// TIA Portal V20 export
FUNCTION "04 T1-A ARUNC Transitions" : Void   // FC1402, LAD
TITLE = TRANSITIONS
{ S7_Optimized_Access := 'TRUE' }
// stored: AutoNumber false, SetENOAutomatically false
   VAR_TEMP
      Aux_real : Real;
   END_VAR
BEGIN

REGION Network 1: ============ TRANSITIONS ============
END_REGION

REGION Network 2: Transitions - Zone Status
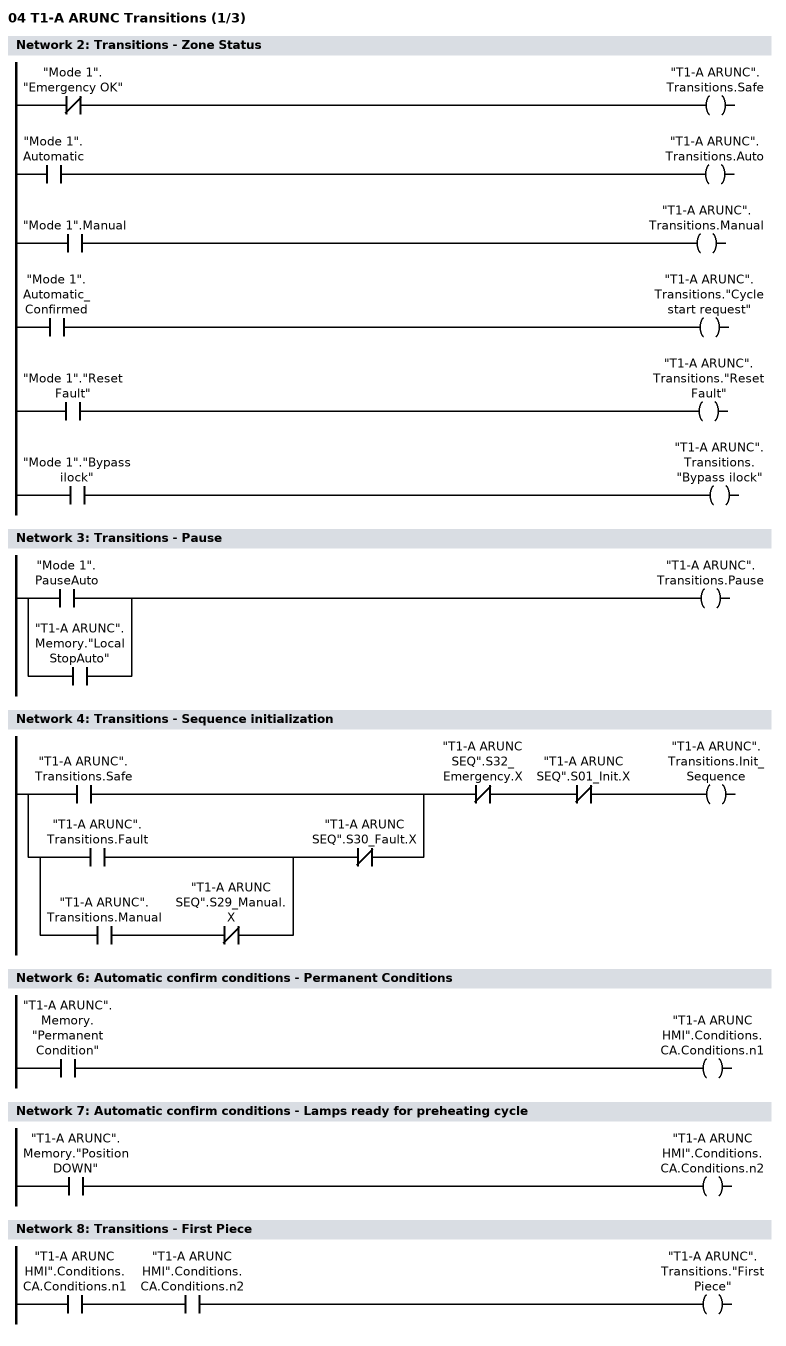
   RUNG wire#powerrail
      I_Contact( "Mode 1"."Emergency OK" )
      Coil( "T1-A ARUNC".Transitions.Safe )
   END_RUNG
   RUNG wire#powerrail
      Contact( "Mode 1".Automatic )
      Coil( "T1-A ARUNC".Transitions.Auto )
   END_RUNG
   RUNG wire#powerrail
      Contact( "Mode 1".Manual )
      Coil( "T1-A ARUNC".Transitions.Manual )
   END_RUNG
   RUNG wire#powerrail
      Contact( "Mode 1".Automatic_Confirmed )
      Coil( "T1-A ARUNC".Transitions."Cycle start request" )
   END_RUNG
   RUNG wire#powerrail
      Contact( "Mode 1"."Reset Fault" )
      Coil( "T1-A ARUNC".Transitions."Reset Fault" )
   END_RUNG
   RUNG wire#powerrail
      Contact( "Mode 1"."Bypass ilock" )
      Coil( "T1-A ARUNC".Transitions."Bypass ilock" )
   END_RUNG
   // the same network as SCL:
   "T1-A ARUNC".Transitions.Safe := NOT "Mode 1"."Emergency OK";
   "T1-A ARUNC".Transitions.Auto := "Mode 1".Automatic;
   "T1-A ARUNC".Transitions.Manual := "Mode 1".Manual;
   "T1-A ARUNC".Transitions."Cycle start request" := "Mode 1".Automatic_Confirmed;
   "T1-A ARUNC".Transitions."Reset Fault" := "Mode 1"."Reset Fault";
   "T1-A ARUNC".Transitions."Bypass ilock" := "Mode 1"."Bypass ilock";
END_REGION

REGION Network 3: Transitions - Pause
   RUNG wire#powerrail
      Contact( "Mode 1".PauseAuto )
      wire#w1
      Coil( "T1-A ARUNC".Transitions.Pause )
   END_RUNG
   RUNG wire#powerrail
      Contact( "T1-A ARUNC".Memory."Local StopAuto" )
   END_RUNG wire#w1
   // the same network as SCL:
   "T1-A ARUNC".Transitions.Pause := "Mode 1".PauseAuto OR "T1-A ARUNC".Memory."Local StopAuto";
END_REGION

REGION Network 4: Transitions - Sequence initialization
   RUNG wire#powerrail
      Contact( "T1-A ARUNC".Transitions.Safe )
      wire#w1
      I_Contact( "T1-A ARUNC SEQ".S32_Emergency.X )
      I_Contact( "T1-A ARUNC SEQ".S01_Init.X )
      Coil( "T1-A ARUNC".Transitions.Init_Sequence )
   END_RUNG
   RUNG wire#powerrail
      Contact( "T1-A ARUNC".Transitions.Fault )
      wire#w2
      I_Contact( "T1-A ARUNC SEQ".S30_Fault.X )
   END_RUNG wire#w1
   RUNG wire#powerrail
      Contact( "T1-A ARUNC".Transitions.Manual )
      I_Contact( "T1-A ARUNC SEQ".S29_Manual.X )
   END_RUNG wire#w2
   // the same network as SCL:
   "T1-A ARUNC".Transitions.Init_Sequence := ("T1-A ARUNC".Transitions.Safe OR (("T1-A ARUNC".Transitions.Fault OR ("T1-A ARUNC".Transitions.Manual AND NOT "T1-A ARUNC SEQ".S29_Manual.X)) AND NOT "T1-A ARUNC SEQ".S30_Fault.X)) AND NOT "T1-A ARUNC SEQ".S32_Emergency.X AND NOT "T1-A ARUNC SEQ".S01_Init.X;
END_REGION

REGION Network 5: ============ AUTOMATIC CONFIRM CONDITIONS - 1ST PIECE ============
END_REGION

REGION Network 6: Automatic confirm conditions - Permanent Conditions
   RUNG wire#powerrail
      Contact( "T1-A ARUNC".Memory."Permanent Condition" )
      Coil( "T1-A ARUNC HMI".Conditions.CA.Conditions.n1 )
   END_RUNG
   // the same network as SCL:
   "T1-A ARUNC HMI".Conditions.CA.Conditions.n1 := "T1-A ARUNC".Memory."Permanent Condition";
END_REGION

REGION Network 7: Automatic confirm conditions - Lamps ready for preheating cycle
   RUNG wire#powerrail
      Contact( "T1-A ARUNC".Memory."Position DOWN" )
      Coil( "T1-A ARUNC HMI".Conditions.CA.Conditions.n2 )
   END_RUNG
   // the same network as SCL:
   "T1-A ARUNC HMI".Conditions.CA.Conditions.n2 := "T1-A ARUNC".Memory."Position DOWN";
END_REGION

REGION Network 8: Transitions - First Piece
   RUNG wire#powerrail
      Contact( "T1-A ARUNC HMI".Conditions.CA.Conditions.n1 )
      Contact( "T1-A ARUNC HMI".Conditions.CA.Conditions.n2 )
      Coil( "T1-A ARUNC".Transitions."First Piece" )
   END_RUNG
   // the same network as SCL:
   "T1-A ARUNC".Transitions."First Piece" := "T1-A ARUNC HMI".Conditions.CA.Conditions.n1 AND "T1-A ARUNC HMI".Conditions.CA.Conditions.n2;
END_REGION

REGION Network 9: Transitions - Piece presence
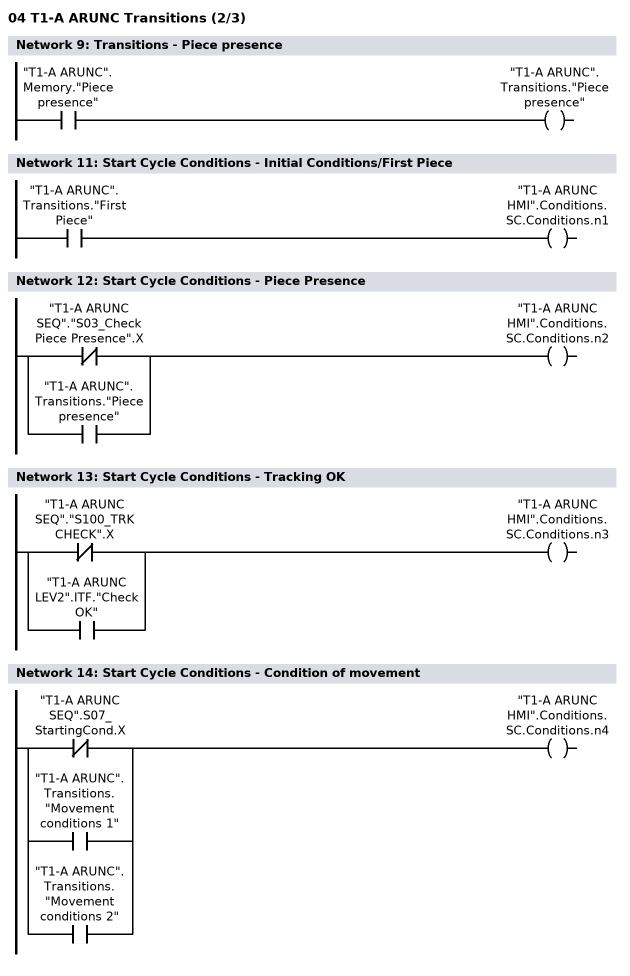
   RUNG wire#powerrail
      Contact( "T1-A ARUNC".Memory."Piece presence" )
      Coil( "T1-A ARUNC".Transitions."Piece presence" )
   END_RUNG
   // the same network as SCL:
   "T1-A ARUNC".Transitions."Piece presence" := "T1-A ARUNC".Memory."Piece presence";
END_REGION

REGION Network 10: ============ START CYCLE CONDITIONS ============
END_REGION

REGION Network 11: Start Cycle Conditions - Initial Conditions/First Piece
   RUNG wire#powerrail
      Contact( "T1-A ARUNC".Transitions."First Piece" )
      Coil( "T1-A ARUNC HMI".Conditions.SC.Conditions.n1 )
   END_RUNG
   // the same network as SCL:
   "T1-A ARUNC HMI".Conditions.SC.Conditions.n1 := "T1-A ARUNC".Transitions."First Piece";
END_REGION

REGION Network 12: Start Cycle Conditions - Piece Presence
   RUNG wire#powerrail
      I_Contact( "T1-A ARUNC SEQ"."S03_Check Piece Presence".X )
      wire#w1
      Coil( "T1-A ARUNC HMI".Conditions.SC.Conditions.n2 )
   END_RUNG
   RUNG wire#powerrail
      Contact( "T1-A ARUNC".Transitions."Piece presence" )
   END_RUNG wire#w1
   // the same network as SCL:
   "T1-A ARUNC HMI".Conditions.SC.Conditions.n2 := NOT "T1-A ARUNC SEQ"."S03_Check Piece Presence".X OR "T1-A ARUNC".Transitions."Piece presence";
END_REGION

REGION Network 13: Start Cycle Conditions - Tracking OK
   RUNG wire#powerrail
      I_Contact( "T1-A ARUNC SEQ"."S100_TRK CHECK".X )
      wire#w1
      Coil( "T1-A ARUNC HMI".Conditions.SC.Conditions.n3 )
   END_RUNG
   RUNG wire#powerrail
      Contact( "T1-A ARUNC LEV2".ITF."Check OK" )
   END_RUNG wire#w1
   // the same network as SCL:
   "T1-A ARUNC HMI".Conditions.SC.Conditions.n3 := NOT "T1-A ARUNC SEQ"."S100_TRK CHECK".X OR "T1-A ARUNC LEV2".ITF."Check OK";
END_REGION

REGION Network 14: Start Cycle Conditions - Condition of movement
   RUNG wire#powerrail
      I_Contact( "T1-A ARUNC SEQ".S07_StartingCond.X )
      wire#w1
      Coil( "T1-A ARUNC HMI".Conditions.SC.Conditions.n4 )
   END_RUNG
   RUNG wire#powerrail
      Contact( "T1-A ARUNC".Transitions."Movement conditions 1" )
   END_RUNG wire#w1
   RUNG wire#powerrail
      Contact( "T1-A ARUNC".Transitions."Movement conditions 2" )
   END_RUNG wire#w1
   // the same network as SCL:
   "T1-A ARUNC HMI".Conditions.SC.Conditions.n4 := NOT "T1-A ARUNC SEQ".S07_StartingCond.X OR "T1-A ARUNC".Transitions."Movement conditions 1" OR "T1-A ARUNC".Transitions."Movement conditions 2";
END_REGION

REGION Network 15: Start Cycle Conditions - next machine consent
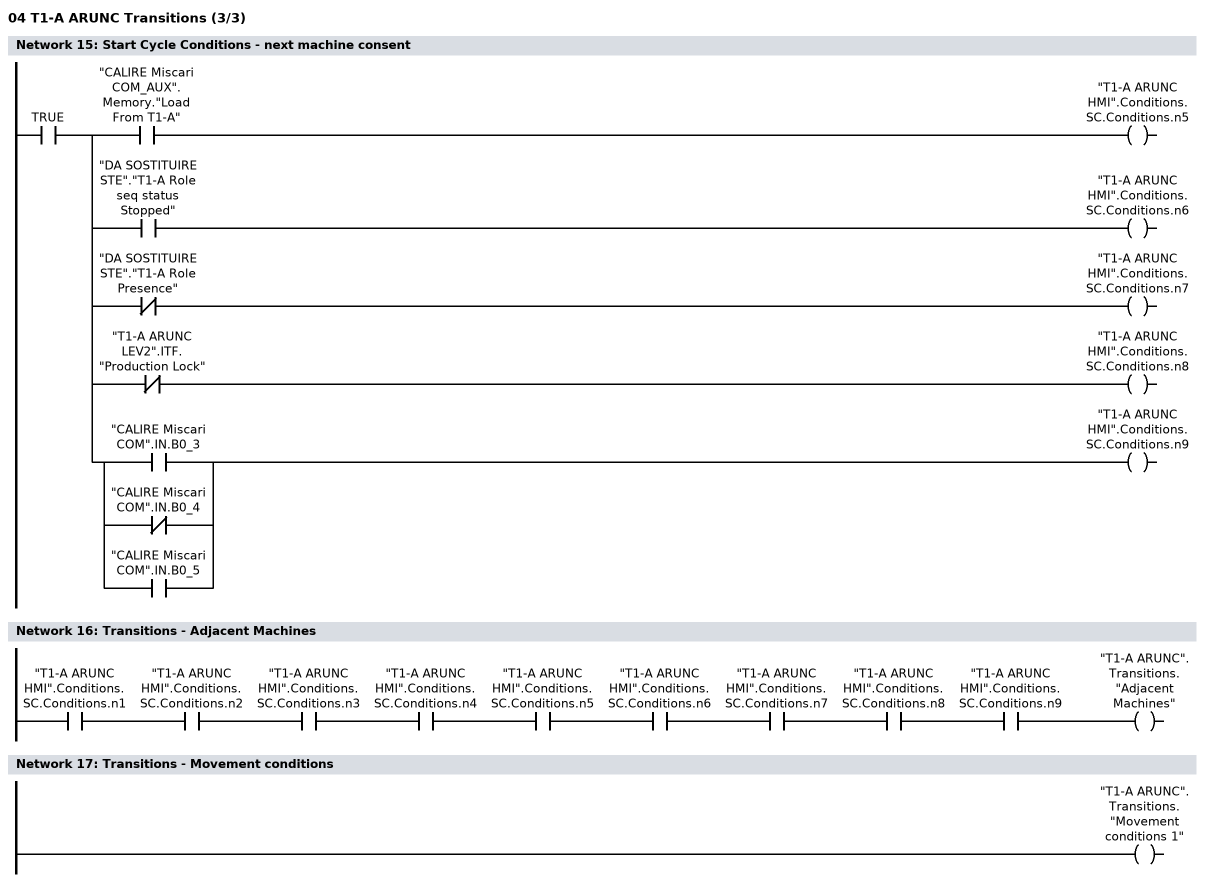
   RUNG wire#powerrail
      Contact( TRUE )
      wire#w1
      Contact( "CALIRE Miscari COM_AUX".Memory."Load From T1-A" )
      Coil( "T1-A ARUNC HMI".Conditions.SC.Conditions.n5 )
   END_RUNG
   RUNG wire#w1
      Contact( "DA SOSTITUIRE STE"."T1-A Role seq status Stopped" )
      Coil( "T1-A ARUNC HMI".Conditions.SC.Conditions.n6 )
   END_RUNG
   RUNG wire#w1
      I_Contact( "DA SOSTITUIRE STE"."T1-A Role Presence" )
      Coil( "T1-A ARUNC HMI".Conditions.SC.Conditions.n7 )
   END_RUNG
   RUNG wire#w1
      I_Contact( "T1-A ARUNC LEV2".ITF."Production Lock" )
      Coil( "T1-A ARUNC HMI".Conditions.SC.Conditions.n8 )
   END_RUNG
   RUNG wire#w1
      Contact( "CALIRE Miscari COM".IN.B0_3 )
      wire#w2
      Coil( "T1-A ARUNC HMI".Conditions.SC.Conditions.n9 )
   END_RUNG
   RUNG wire#w1
      I_Contact( "CALIRE Miscari COM".IN.B0_4 )
   END_RUNG wire#w2
   RUNG wire#w1
      Contact( "CALIRE Miscari COM".IN.B0_5 )
   END_RUNG wire#w2
   // the same network as SCL:
   "T1-A ARUNC HMI".Conditions.SC.Conditions.n5 := TRUE AND "CALIRE Miscari COM_AUX".Memory."Load From T1-A";
   "T1-A ARUNC HMI".Conditions.SC.Conditions.n6 := TRUE AND "DA SOSTITUIRE STE"."T1-A Role seq status Stopped";
   "T1-A ARUNC HMI".Conditions.SC.Conditions.n7 := TRUE AND NOT "DA SOSTITUIRE STE"."T1-A Role Presence";
   "T1-A ARUNC HMI".Conditions.SC.Conditions.n8 := TRUE AND NOT "T1-A ARUNC LEV2".ITF."Production Lock";
   "T1-A ARUNC HMI".Conditions.SC.Conditions.n9 := TRUE AND ("CALIRE Miscari COM".IN.B0_3 OR NOT "CALIRE Miscari COM".IN.B0_4 OR "CALIRE Miscari COM".IN.B0_5);
END_REGION

REGION Network 16: Transitions - Adjacent Machines
   RUNG wire#powerrail
      Contact( "T1-A ARUNC HMI".Conditions.SC.Conditions.n1 )
      Contact( "T1-A ARUNC HMI".Conditions.SC.Conditions.n2 )
      Contact( "T1-A ARUNC HMI".Conditions.SC.Conditions.n3 )
      Contact( "T1-A ARUNC HMI".Conditions.SC.Conditions.n4 )
      Contact( "T1-A ARUNC HMI".Conditions.SC.Conditions.n5 )
      Contact( "T1-A ARUNC HMI".Conditions.SC.Conditions.n6 )
      Contact( "T1-A ARUNC HMI".Conditions.SC.Conditions.n7 )
      Contact( "T1-A ARUNC HMI".Conditions.SC.Conditions.n8 )
      Contact( "T1-A ARUNC HMI".Conditions.SC.Conditions.n9 )
      Coil( "T1-A ARUNC".Transitions."Adjacent Machines" )
   END_RUNG
   // the same network as SCL:
   "T1-A ARUNC".Transitions."Adjacent Machines" := "T1-A ARUNC HMI".Conditions.SC.Conditions.n1 AND "T1-A ARUNC HMI".Conditions.SC.Conditions.n2 AND "T1-A ARUNC HMI".Conditions.SC.Conditions.n3 AND "T1-A ARUNC HMI".Conditions.SC.Conditions.n4 AND "T1-A ARUNC HMI".Conditions.SC.Conditions.n5 AND "T1-A ARUNC HMI".Conditions.SC.Conditions.n6 AND "T1-A ARUNC HMI".Conditions.SC.Conditions.n7 AND "T1-A ARUNC HMI".Conditions.SC.Conditions.n8 AND "T1-A ARUNC HMI".Conditions.SC.Conditions.n9;
END_REGION

REGION Network 17: Transitions - Movement conditions
   RUNG wire#powerrail
      Coil( "T1-A ARUNC".Transitions."Movement conditions 1" )
   END_RUNG
   // the same network as SCL:
   "T1-A ARUNC".Transitions."Movement conditions 1" := TRUE;
END_REGION
END_FUNCTION
